                // setpoint for melt temperature control
                //--------------------------------------
                "AC".SET_MLT_1_TMP    :=    "PAR_MAIN".DI_TMP_DIPPING;

                // time till end of this step
                // --------------------------
                "APC".ACT_TME_STE := #par_time - "APC".TI[0];

                //end of step
                //-----------
                IF ("APC".TI[0] > #par_time) THEN
                    //setpoint calculation for temperature decrement
                    //----------------------------------------------
                    "AC".SET_HTR_1_TMP     :=    #htr_1_tmp_before_gap - "PAR_MAIN".DI_TMP_DEC_HTR_1;
                    #end_of_step[0] := true;
                END_IF;

                #next_step[0] := 950;


   //-step-950--level--0--------------------------------------------------------------                                                  
   //            DI: wait time after temperature decrement
   //---------------------------------------------------------------------------------                                                 
            950 :
                 IF #next_step[0] = #active_step[0] THEN   
                     "APC".TI[0] := 0;                     // start step time
                 END_IF;

                 //end of step
                 //-----------
                 IF ("APC".TI[0] > 5) THEN
                     #end_of_step[0] := true;
                 END_IF;

                 #next_step[0] := 1000;


   //-step-1000--level--0-------------------------------------------------------------                                                 
   //            DI: start neck process
   //---------------------------------------------------------------------------------                                                 
           1000 :                                                  
                 IF #next_step[0] = #active_step[0] THEN
                   "APC".OP_MSG := "OP_MSG".BLANK;
                   "DC".MOD_NE := TRUE;                           // switch to neck 
                 END_IF;

                 #next_step[0] := 1000;                        // E N D


   //-error------level--0---------------------------------------------------(error in level 0)-------------
       ELSE:                                                        
           //error code                                                //do error code
           ;        
   //------------------------------------------------------------------------------------------------------
       END_CASE;

       //check if calculated weight of grown body is changed
       //---------------------------------------------------
       IF ("KYA".CALC_WGT_GRW_XT <> #prv_calc_wgt_grw_xt) THEN
           #xt_wgt_chgd     :=  true;

       END_IF;

       //calculation length of next body
       //-------------------------------
       IF (#xt_wgt_chgd OR NOT #xt_lgh_calc_done) THEN 

           //call calculation of 2nd body length
           //-----------------------------------
           "CM_CALC_NEXT_BY" (dia            := "PAR_XT_DIA".PAR[7, 1],       
                            xt_wgt_cor     := ("KYA".CALC_WGT_GRW_XT - #prv_calc_wgt_grw_xt),
                            rm_mlt         := "CNF".RM_MLT_AFT_PRC);

           #prv_calc_wgt_grw_xt :=  "KYA".CALC_WGT_GRW_XT;
           #xt_lgh_calc_done    :=  true;
           #xt_wgt_chgd         :=  false;

       END_IF;

       #start_previous  := #start;                                   //save start input for next call 
       #cont_previous   := "APC".CONT;                                //save cont input for next call 
       #resume_previous := "APC".RESUME;                              //save resume input for next call
       #jump_previous   := "APC".JUMP;                                //save jump input for next call
       #single_previous := "APC".SINGLE;                              //save single input for next call
END_FUNCTION_BLOCK

FUNCTION_BLOCK "AM_NE"   // FB199, SCL
{ S7_Optimized_Access := 'FALSE' }
VERSION : 0.0
// --------------------------------------------------------------------------------
//     program     :    AM_NE
//     description :    apc neck module  
//     name        :    D. Bruess
//     date        :    25.11.99
// 
//     revision    :    change default rotation direction: xtal= ccw and cruc= cw
//     name        :    G. Eibelsh鋟ser
//     date        :    26.04.00
// 
//     revision    :    
//     name        :    
//     date        :    
//                     (c)CGS
//     --------------------------------------------------------------------------------
   VAR_INPUT
      start : Bool;   // start sequence, activate step 10 (impulse triggered)
   END_VAR
   VAR
      start_previous : Bool;   // start input value of last call
      cont_previous : Bool;   // cont input value of last call
      resume_previous : Bool;   // resume input value of last call
      jump_previous : Bool;   // jump input value of last call
      single_previous : Bool;   // single input value of last call
      active_step : Array[0..7] of Int;   // active step number for sequence level 0..7
      next_step : Array[0..7] of Int;   // next step number for sequence level 0..7
      hold_step : Array[0..7] of Int;   // step number of step on hold
      end_of_step : Array[0..7] of Bool;   // active step is done flag for sequence 0..7
      EndOfStep : Bool;   // default value for active step is done flag
      cont_enable : Array[0..7] of Bool;   // enable continue function
      ContEnable : Bool;   // default value for enable continue function
      ne_end : Bool;   // neck end flag
      xt_pos_at_start : Real;   // crystal position at start of neck
      xt_dia_at_start : Real;   // crystal diameter at start
      xt_dia_end_slope1 : Real;   // crystal diameter at end of slope 1
      xt_dia_end_slope2 : Real;   // crystal diameter at end of slope 2
      ini_ne_len : Real;   // initial stable neck length
   END_VAR
BEGIN


       "APC".STATUS := "APC".NECK;                                     // set apc status               

       "AM_SEQUENCE_CTL" (start_p            := #start,               // control sequence
                        start_previous_p   := #start_previous,
                        cont_previous_p    := #cont_previous, 
                        resume_previous_p  := #resume_previous,
                        jump_previous_p    := #jump_previous,
                        single_previous_p  := #single_previous,
                        active_step_p      := #active_step, 
                        next_step_p        := #next_step,
                        hold_step_p        := #hold_step, 
                        end_of_step_p      := #end_of_step, 
                        cont_enable_p      := #cont_enable); 

       //Set the "Oxidation valve" in all Phases
       "DC".V21_OP:= DINT_TO_BOOL(REAL_TO_DINT("PAR_MAIN".NE_V21_OPEN));

       CASE #active_step[0] OF    //sequence level_0
   //step--0-----level--0-------------------------------------------------off--(sequence off)--------------
           0    :                                                  
                #next_step[0] := 0;

   //step--1-----level--0-------------------------------------------------hold-(test sequence)-------------
           1   :                                                       
               IF #next_step[0] = #active_step[0] THEN                   //init step     
                   //init code
                   ; 
               END_IF;

               //step code                                             //do step
               ;

   //-step-10----level--0----------------------------------------------main-(start sequence)---------------                                                 

   //-step-10----level--0-------------------------------------------------------------                                                 
   //            NE: init neck sequence
   //---------------------------------------------------------------------------------                                                 
           10  :                                                     

               // init vacuum system
               // ------------------
               "DC".V1_OP    := TRUE;                         // open V1
               "DC".V3_OP    := FALSE;
               "DC".V4_OP    := FALSE;
               "DC".V5_OP    := TRUE;                         // open V5
               "DC".V6_OP    := FALSE;
               "DC".V8_OP    := FALSE;
               "DC".V11_OP   := FALSE;
               "DC".V11_CL   := TRUE;
               "DC".V12_OP   := FALSE;
               "DC".V13_OP   := FALSE;
               "DC".V20_OP   := FALSE;
               "DC".V22_OP   := FALSE;
               "DC".V24_OP   := FALSE;
               "DC".P1_ON    := TRUE;                         // start main pump
               "DC".P3_ON    := FALSE;
               "DC".V3_4_OP  := FALSE;
               "DC".V1_1_REL := FALSE;

               "DC".V3_2_OP := FALSE;                      // vacuum valve feeder

               "DC".V1_OPEN_REQ   := FALSE;                // only EKZ 2700
               "DC".V1_CLOSE_REQ  := FALSE;


               // init drives
               // -----------
               "DC".XT_LFT_UP := TRUE;                     // crystal lift up
               "DC".XT_LFT_DN := FALSE;
               "DC".XT_LFT_FST := FALSE;
               "DC".XT_ROT_CW := "BM_ROT_DRV_DIR_DB".ROT_DIR;            //1 = cw
               "DC".XT_ROT_CCW := NOT "BM_ROT_DRV_DIR_DB".ROT_DIR;       //0 = ccw


               "DC".CR_LFT_UP := FALSE;                    // crucible lift up
               "DC".CR_LFT_DN := FALSE;
               "DC".CR_LFT_FST := FALSE;
               "DC".CR_ROT_CW := NOT "BM_ROT_DRV_DIR_DB".ROT_DIR;        //0 = cw
               "DC".CR_ROT_CCW := "BM_ROT_DRV_DIR_DB".ROT_DIR;           //1 = ccw


               "AC".SET_XT_SPD := "KYA".SET_XT_SPD;
               "AC".SET_XT_ROT := "KYA".SET_XT_ROT;
               "AC".SET_CR_SPD := 0.0;
               "AC".SET_CR_ROT := "KYA".SET_CR_ROT;

               // init heater
               // -----------
               "DC".HTR_1_ON := TRUE;                     // heater on
               "DC".HTR_2_ON := TRUE;
               "DC".HTR_3_ON := FALSE;

               // AC.SET_HTR_1_PWR := 0.0;                 do not set, loop is on
               // AC.SET_HTR_2_PWR := 0.0;
               // AC.SET_HTR_3_PWR := 0.0;

               //mobile feeder
               //-------------
               "DC".MOB_FDR_MVE_IN_SEQ_ON    :=  FALSE;
               IF ("LT".MOB_FDR_DCK_DONE AND ("DV".FDG_MVE_IN_SEQ_DONE OR NOT "DV".FDG_MVE_OUT_SEQ_DONE)) THEN 
                   "DC".MOB_FDR_MVE_OUT_SEQ_ON   :=  TRUE;
               ELSE
                   "DC".MOB_FDR_MVE_OUT_SEQ_ON   :=  FALSE;
               END_IF;
               "DC".MOB_FDR_VIB_ON           :=  FALSE;
               "FLT".MOB_FDR_NOT_DCK         :=  FALSE;
               "FLT".MOB_FDR_STP_PARA        :=  FALSE;

               // init magnet
               // -----------
               "DC".MAG_ON := ("AC".SET_MAG_1_CUR > 0.0);                       

               "AC".SET_MAG_1_CUR := "KYA".SET_MAG_1_CUR;
               "AC".SET_MAG_2_CUR := "KYA".SET_MAG_2_CUR;

               // init control loops
               // ------------------
               "DC".CTL_DIA_ON := FALSE;                   // all control loops off
               "DC".CTL_GRW_RTE_ON := FALSE;
               "DC".CTL_PULL_RTE_ON := FALSE;
               "DC".CTL_CRUC_ROT_ON := FALSE;
               "DC".CTL_MLT_LVL_ON := FALSE;
               "DC".CTL_MLT_1_TMP_ON := FALSE;
               "DC".CTL_MLT_2_TMP_ON := FALSE;
               "DC".CTL_MLT_DRIFT_ON := FALSE;
               "DC".CTL_GAP_ON       := FALSE;
               "DC".CTL_HTR_1_TMP_ON := TRUE;              // heater temp loop on
               //  DC.CTL_HTR_2_TMP_ON := TRUE;

               "DC".SET_HTR_1_TMP_ABS := FALSE;            // enable inc functions
               "DC".SET_HTR_2_PWR_ABS := FALSE;


               "DC".CTL_PRS_ON := TRUE;                    // pressure control on

               "DC".CTL_SI_FDR_ON := FALSE;
               "DC".CTL_DOP_FDR_ON := FALSE;

               "DV".TRANS_SH_BY_FLAG := FALSE;
               "DV".START_SH_FLAG    := FALSE;

               "AC".SET_XT_DIA := 0.0;
               "AC".SET_GRW_RTE := 0.0;
               "AC".SET_AVG_SPD := 0.0;
               "AC".SET_AVG_CRUC_ROT := 0.0;
               "AC".SET_MLT_LVL_LSR := 0.0;
               "AC".SET_MLT_1_TMP := 0.0;
               "AC".SET_MLT_2_TMP := 0.0;

               // init measurement system
               // -----------------------
               "DC".CAM_ISP_ON   :=  TRUE;      //inspection on
               "DC".CAM_INIT     :=  FALSE;
               "DC".CAM_MLT      :=  FALSE;
               "DC".CAM_DIP      :=  FALSE;
               "DC".CAM_DIA      :=  TRUE;
               "DC".CAM_SEL_1    :=  TRUE;
               "DC".CAM_SEL_2    :=  FALSE;

               "DV".THR_CALC_DISABLED  := TRUE;      //threshold calculation in this step is disabled


               "DC".LSR_ON := ("PAR_MAIN".BY_LSR_LVL_CTL_ON = 1.0);    // laser on/off (parameter comes from body mode)
               "DC".MCC_ON := FALSE;                                 // melt contact control off
               "DC".MCC_TST_ON := FALSE;

               // init Si feeder system
               // ---------------------
               "DC".SI_FDR_ON := FALSE;                              // feeder off
               "DC".DOP_FDR_ON := FALSE;

               "AC".SET_FDR_SI := 0.0;
               "AC".SET_FDR_DOP := 0.0;

               // init lamp on control cabinet
               // ----------------------------
               "DV".LMP_OR := false;

               // save start position, reset length
               // ---------------------------------
               #xt_pos_at_start := "AV".ACT_XT_POS;
               "AV".ACT_XT_LEN_PRC := 0.0; 
               "AV".ACT_XT_LEN := 0.0;

               // calculate all setpoints 
               // -----------------------
               "AM_PAR_FNC_NE" (act_x_value := 0.0);
               "AC".SET_XT_DIA := "AV".ACT_XT_DIA;           // setpoint = act. diameter 

               // enable automatic mode
               // ---------------------
               "DC".MOD_AUT_ENB := TRUE;

               #end_of_step[0] := true;                            
               #next_step[0] := 100;

   //-step-100---level--0-------------------------------------------------------------                                                 
   //            NE: wait for automatic mode
   //---------------------------------------------------------------------------------                                                 
           100 :                                                     
               IF #next_step[0] = #active_step[0] THEN
                   "APC".OP_MSG := "OP_MSG".WAIT_FOR_AUTO;                                                  
               END_IF;

               // do not count the length while waiting for automatic
               // ---------------------------------------------------
               #xt_pos_at_start := "AV".ACT_XT_POS;
               "AV".ACT_XT_LEN_PRC := 0.0; 
               "AV".ACT_XT_LEN := 0.0;

               // calculate all setpoints 
               // -----------------------
               "AM_PAR_FNC_NE" (act_x_value := 0.0);
               "AC".SET_XT_DIA := "AV".ACT_XT_DIA;           // setpoint = act. diameter 

               IF "APC".AUTOMATIC = TRUE THEN                     // automatic mode ?
                   #end_of_step[0] := true;                            
               END_IF;                                    
               #next_step[0] := 200;


   //-step-200---level--0-------------------------------------------------------------                                                 
   //            NE: start time
   //---------------------------------------------------------------------------------                                                 
           200 :                                                     
               "APC".ACT_TME_PROC := 0;                           // start process time
               "APC".ACT_TME_STE := 0;                            // reset time of step
               "APC".TI[0] := 0;                                  // start waiting time
               "APC".OP_MSG := "OP_MSG".BLANK;                                                  

               //init total length calculation
               //-----------------------------
               "DV".NE_RESTART   :=  TRUE;

               #end_of_step[0] := true;                            
               #next_step[0] := 300;

   //-step-300---level--0-------------------------------------------------------------                                                 
   //            NE: do initial temp. inc. and wait (const speed, no dia. control)
   //---------------------------------------------------------------------------------                                                 
           300 :                                                     
               IF #next_step[0] = #active_step[0] THEN                       
                   //display initial temperature and power setpoints
                   //-----------------------------------------------
                   "DIS".HTR_1_TMP_SET_PHA_STR   :=  "CTL".SET_HTR_1_TMP;
                   "DIS".HTR_2_PWR_SET_PHA_STR   :=  "CTL".SET_HTR_2_PWR;
                   // do heater inc.
                   // --------------
                   "DC".RSTRT_HTR_1_TMP_INC      := TRUE;
                   "DC".RSTRT_HTR_2_PWR_INC      := TRUE;
                   "AC".SET_HTR_1_TMP_INC        := "AV".SET_HTR_1_TMP_INC;
                   "AC".SET_HTR_2_PWR_INC        := "AV".SET_HTR_2_PWR_INC;

                   "AV".SET_DIP_TMP              := "CTL".SET_HTR_1_TMP;           //store heater temp setpoint (used in removal)
                   "APC".OP_MSG                  := "OP_MSG".BY_WAIT_TILL_DIA_CTL;

               END_IF;

               // setpoint magnet
               // ---------------
               "DC".MAG_ON := ("AC".SET_MAG_1_CUR > 0.0);

               "AC".SET_MAG_1_CUR := "AV".SET_MAG_1_CUR;
               "AC".SET_MAG_2_CUR := "AV".SET_MAG_1_CUR * "AV".SET_MAG_RATIO_CUR;


               // calculate actual length
               // -----------------------
               "AM_CALC_LENGTH" (start_pos := #xt_pos_at_start,
                               actual_pos := "AV".ACT_XT_POS,
                               total_len := -1.0,              // % not calculated
                               actual_len => "AV".ACT_XT_LEN,
                               actual_len_prc => "AV".ACT_XT_LEN_PRC);


               // calculate all setpoints for this step
               // -------------------------------------                                      
               "AM_PAR_FNC_NE" (act_x_value := 0.0);
               "AC".SET_XT_DIA := "AV".ACT_XT_DIA;         // setpoint = act. diameter 
               "AC".SET_XT_SPD := "AC".SET_AVG_SPD;        // init output diam. control
               "AC".SET_HTR_1_TMP_INC := "AV".SET_HTR_1_TMP_INC;
               "AC".SET_HTR_2_PWR_INC := "AV".SET_HTR_2_PWR_INC;


               // wait time ?
               // -----------
               IF ("APC".TI[0] > 30) THEN
                  #end_of_step[0] := true;
               END_IF;

               #next_step[0] := 400; 


   //-step-400---level--0-------------------------------------------------------------                                                 
   //            NE: grow neck cone (slope 1)
   //---------------------------------------------------------------------------------                                                 
           400 :                                                  
               IF #next_step[0] = #active_step[0] THEN                       
                   // start time for slope calc.
                   // --------------------------
                   "APC".TI[0] := 0;

                   // save start diameter
                   // -------------------
                   #xt_dia_at_start := "AV".ACT_XT_DIA;
                   "AC".SET_XT_DIA   := "AV".ACT_XT_DIA;           // setpoint = act. diameter 

                   // diameter and av. speed control on
                   // ---------------------------------
                   "DC".CTL_DIA_ON       := TRUE;
                   "DC".CTL_PULL_RTE_ON  := TRUE;

                   "APC".OP_MSG := "OP_MSG".NE_DIA_REDUCTION1;
               END_IF;

               // setpoint magnet
               // ---------------
               "DC".MAG_ON := ("AC".SET_MAG_1_CUR > 0.0);

               "AC".SET_MAG_1_CUR := "AV".SET_MAG_1_CUR;
               "AC".SET_MAG_2_CUR := "AV".SET_MAG_1_CUR * "AV".SET_MAG_RATIO_CUR;

               // calculate actual length
               // -----------------------
               "AM_CALC_LENGTH" (start_pos      := #xt_pos_at_start,
                               actual_pos     := "AV".ACT_XT_POS,
                               total_len      := -1.0,              // % not calculated
                               actual_len     => "AV".ACT_XT_LEN,
                               actual_len_prc => "AV".ACT_XT_LEN_PRC);

               // calculate all setpoints for this step
               // -------------------------------------                                      
               "AM_PAR_FNC_NE" (act_x_value := 0.0);           // use first line
               #xt_dia_end_slope1 := "PAR_XT_DIA".PAR["APC".NECK, 1]
                                                  + "CNF".NECK_DELTA_SLOPE_1;
               #xt_dia_end_slope2 := "PAR_XT_DIA".PAR["APC".NECK, 1];


               "AM_CALC_NECK_DIA" (d0  := #xt_dia_at_start,
                                 dend:= #xt_dia_end_slope2,
                                 t   := INT_TO_REAL("APC".TI[0]),
                                 ddt := "CNF".NECK_SLOPE_1,
                                 dia => "AC".SET_XT_DIA);

               // heater temp/power inc.
               // ----------------------
               "AC".SET_HTR_1_TMP_INC := "AV".SET_HTR_1_TMP_INC;
               "AC".SET_HTR_2_PWR_INC := "AV".SET_HTR_2_PWR_INC;

               // melt contact control
               // --------------------   
               "DC".MCC_ON := ("PAR_MAIN".NE_MLT_CONTACT_CTL = 1.0);        


               // diameter setpoint below (final diam. + delta) ?
               // -----------------------------------------------
               IF ("AC".SET_XT_DIA < #xt_dia_end_slope1) THEN    
                   #end_of_step[0] := true;                            
               END_IF;
               #next_step[0] := 500; 


   //-step-500---level--0-------------------------------------------------------------                                                 
   //            NE: grow neck cone (slope 2)
   //---------------------------------------------------------------------------------                                                 
           500 :                                                  
               IF #next_step[0] = #active_step[0] THEN                       
                   // start time for slope calc.
                   // --------------------------
                   "APC".TI[0] := 0;

                   // save start diameter setpoint
                   // ----------------------------
                   #xt_dia_at_start := "AC".SET_XT_DIA;

                   "APC".OP_MSG := "OP_MSG".NE_DIA_REDUCTION2;
               END_IF;

               // setpoint magnet
               // ---------------
               "DC".MAG_ON := ("AC".SET_MAG_1_CUR > 0.0);

               "AC".SET_MAG_1_CUR := "AV".SET_MAG_1_CUR;
               "AC".SET_MAG_2_CUR := "AV".SET_MAG_1_CUR * "AV".SET_MAG_RATIO_CUR;


               // calculate actual length
               // -----------------------
               "AM_CALC_LENGTH" (start_pos := #xt_pos_at_start,
                               actual_pos := "AV".ACT_XT_POS,
                               total_len := -1.0,              // % not calculated
                               actual_len => "AV".ACT_XT_LEN,
                               actual_len_prc => "AV".ACT_XT_LEN_PRC);

               // calculate all setpoints for this step
               // -------------------------------------                                      
               "AM_PAR_FNC_NE" (act_x_value := 0.0);           // use first line
               #xt_dia_end_slope1 := "PAR_XT_DIA".PAR["APC".NECK, 1]
                                                  + "CNF".NECK_DELTA_SLOPE_1;
               #xt_dia_end_slope2 := "PAR_XT_DIA".PAR["APC".NECK, 1];


               "AM_CALC_NECK_DIA" (d0  := #xt_dia_at_start,
                                 dend:= #xt_dia_end_slope2,
                                 t   := INT_TO_REAL("APC".TI[0]),
                                 ddt := "CNF".NECK_SLOPE_2,
                                 dia => "AC".SET_XT_DIA);

               // heater temp/power inc.
               // ----------------------
               "AC".SET_HTR_1_TMP_INC := "AV".SET_HTR_1_TMP_INC;
               "AC".SET_HTR_2_PWR_INC := "AV".SET_HTR_2_PWR_INC;

               // melt contact control
               // --------------------   
               "DC".MCC_ON := ("PAR_MAIN".NE_MLT_CONTACT_CTL = 1.0);        

               // diameter setpoint below final diam. ?
               // -------------------------------------
               IF ("AC".SET_XT_DIA <= #xt_dia_end_slope2) THEN    
                   #end_of_step[0] := true;                            
               END_IF;
               #next_step[0] := 600; 


   //-step-600---level--0-------------------------------------------------------------                                                 
   //            NE: do neck process
   //---------------------------------------------------------------------------------                                                 
           600 :                                                  
               IF #next_step[0] = #active_step[0] THEN                       
                   // save start position, reset length
                   // ---------------------------------
                   #xt_pos_at_start := "AV".ACT_XT_POS;
                   #ini_ne_len      := 0.0;
                   "APC".OP_MSG := "OP_MSG".NE_DIA_CONSTANT;
               END_IF;

               // setpoint magnet
               // ---------------
               "DC".MAG_ON := ("AC".SET_MAG_1_CUR > 0.0);

               "AC".SET_MAG_1_CUR := "AV".SET_MAG_1_CUR;
               "AC".SET_MAG_2_CUR := "AV".SET_MAG_1_CUR * "AV".SET_MAG_RATIO_CUR;

               // heater temp/power inc.
               // ----------------------
               "AC".SET_HTR_1_TMP_INC := "AV".SET_HTR_1_TMP_INC;
               "AC".SET_HTR_2_PWR_INC := "AV".SET_HTR_2_PWR_INC;

               // melt contact control
               // --------------------   
               "DC".MCC_ON := ("PAR_MAIN".NE_MLT_CONTACT_CTL = 1.0);  

               // calculate all setpoints for this step
               // -------------------------------------                                      
               "AM_PAR_FNC_NE" (act_x_value := "AV".ACT_XT_LEN);
               "AC".SET_XT_DIA := "AV".SET_XT_DIA;


                //neck with flexible length (option)
               //----------------------------------
               IF (REAL_TO_INT("PAR_MAIN".NE_LEN_FLX) = 1) THEN  

                   // calculate actual length
                   // -----------------------
                   "AM_CALC_LENGTH" (start_pos       := #xt_pos_at_start,
                                   actual_pos      := "AV".ACT_XT_POS,
                                   total_len       := "PAR_MAIN".NE_MAX_LEN,
                                   actual_len      => "AV".ACT_XT_LEN,
                                   actual_len_prc  => "AV".ACT_XT_LEN_PRC);


                   //reset stable neck length due to diameter or growth deviation, slow pull speed or minimum neck length
                   //----------------------------------------------------------------------------------------------------
                   IF ((("AV".ACT_XT_DIA - "AC".SET_XT_DIA) > "PAR_MAIN".NE_MAX_DEV_DIA)     OR 
                       ("CTL".ACT_GRW_RTE > "PAR_MAIN".NE_MAX_DEV_LAT_GRW)                 OR
                       ("CTL".AVG_XT_SPD < "PAR_MAIN".NE_MIN_XT_SPD)                       OR 
                       ("AV".ACT_XT_LEN <= ("PAR_MAIN".NE_MIN_LEN - "PAR_MAIN".NE_STB_LEN))) THEN

                       #ini_ne_len  :=  "AV".ACT_XT_LEN;
                   END_IF;

                   //calculate stable neck length
                   //----------------------------    
                   "AV".ACT_STB_NE_LEN   :=  "AV".ACT_XT_LEN - #ini_ne_len;

                   IF ("PAR_MAIN".NE_STB_LEN > 0.0) THEN 
                       "AV".ACT_STB_NE_LEN_PRC   :=  "AV".ACT_STB_NE_LEN / "PAR_MAIN".NE_STB_LEN * 100.0;
                   END_IF;

                   //neck end when max. length is reached
                   //------------------------------------ 
                   IF  ("AV".ACT_XT_LEN >= "PAR_MAIN".NE_MAX_LEN) THEN 
                       #ne_end          :=  true;
                       "FLT".NE_MAX_LEN  :=  TRUE;

                   //neck min length reached
                   //-----------------------
                   ELSIF  ("AV".ACT_XT_LEN >= "PAR_MAIN".NE_MIN_LEN) THEN 
                       //check stable neck length
                       //------------------------
                       IF ("AV".ACT_STB_NE_LEN >= "PAR_MAIN".NE_STB_LEN) THEN
                           #ne_end  :=  true;
                       ELSE
                           #ne_end  :=  false;
                       END_IF;
                   ELSE
                       #ne_end  :=  false;
                   END_IF;

                   // check if neck end is reached ?
                   // ------------------------------
                   IF #ne_end THEN    
                       #end_of_step[0] := true;                            
                   END_IF;

               //neck with fixed length (standard)
               //---------------------------------
               ELSE 

                   // calculate actual length
                   // -----------------------
                   "AM_CALC_LENGTH" (start_pos       := #xt_pos_at_start,
                                   actual_pos      := "AV".ACT_XT_POS,
                                   total_len       := "PAR_MAIN".NE_LEN,
                                   actual_len      => "AV".ACT_XT_LEN,
                                   actual_len_prc  => "AV".ACT_XT_LEN_PRC);

                   // 100% of length reached ?
                   // ------------------------
                   IF ("AV".ACT_XT_LEN_PRC >= 100.0) THEN    
                       #end_of_step[0] := true;                            
                   END_IF;

               END_IF;
               #next_step[0] := 700; 


   //-step-700---level--0-------------------------------------------------------------                                                 
   //            NE: start shoulder process
   //---------------------------------------------------------------------------------                                                 
           700 :                                                  
               IF #next_step[0] = #active_step[0] THEN
                   "APC".OP_MSG := "OP_MSG".BLANK;
               END_IF;

               "DC".MOD_SH := TRUE;                               // switch to shoulder 
               #next_step[0] := 700;                             // E N D 



   //-error------level--0---------------------------------------------------(error in level 0)-------------
       ELSE:                                                        
           //error code                                                //do error code
           ;        
   //------------------------------------------------------------------------------------------------------
       END_CASE;

       CASE #active_step[1] OF    //sequence level_1
   //step--0-----level--1-------------------------------------------------off--(sequence off)--------------
           0    :                                                  
                #next_step[1] := 0;

   //step--1-----level--1-------------------------------------------------hold-(test sequence)-------------
           1   :                                                       
               IF #next_step[1] = #active_step[1] THEN                   //init step     
                   //init code
                   ; 
               END_IF;

               //step code                                             //do step
               ;

   //-step-10----level--1----------------------------------------------main-(start sequence)---------------                                                 
           10  :                                                     
               IF #next_step[1] = #active_step[1] THEN                   //init step     
                   //init code 
                   ;                                                  
               END_IF;

               //step code                                             //do step
               ;
               IF #ContEnable = true THEN                               //enable continue function
                   #cont_enable[1] := true;
               END_IF;
               IF #EndOfStep = true THEN                                //define end of step condition
                   #end_of_step[1] := true;                            
               END_IF;                                    
               #next_step[1] := 0;                                      //define next step #
               IF #end_of_step[1] = true THEN                           //do on transition
                   //transition code
                   ;
               END_IF;

   //-step-100---level--1----------------------------------------------name-(remarks)----------------------                                                 
           100 :                                                     
               IF #next_step[1] = #active_step[1] THEN                   //init step     
                   //init code 
                   ;                                                  
               END_IF;

               //step code                                             //do step
               ;
               IF #ContEnable = true THEN                               //enable continue function
                   #cont_enable[1] := true;
               END_IF;
               IF #EndOfStep = true THEN                                //define end of step condition
                   #end_of_step[1] := true;                            
               END_IF;                                    
               #next_step[1] := 0;                                      //define next step #
               IF #end_of_step[1] = true THEN                           //do on transition
                   //transition code
                   ;
               END_IF;

   //-step-200---level--1----------------------------------------------name-(remarks)----------------------                                                 
           200 :                                                     
               IF #next_step[1] = #active_step[1] THEN                   //init step     
                   //init code 
                   ;                                                  
               END_IF;

               //step code                                             //do step
               ;
               IF #ContEnable = true THEN                               //enable continue function
                   #cont_enable[1] := true;
               END_IF;
               IF #EndOfStep = true THEN                                //define end of step condition
                   #end_of_step[1] := true;                            
               END_IF;                                    
               #next_step[1] := 0;                                      //define next step #
               IF #end_of_step[1] = true THEN                           //do on transition
                   //transition code
                   ;
               END_IF;

   //-error------level--1---------------------------------------------------(error in level 1)-------------
       ELSE:                                                        
           //error code                                                //do error code
           ;        
   //------------------------------------------------------------------------------------------------------
       END_CASE;

       CASE #active_step[2] OF    //sequence level_2
   //step--0-----level--2-------------------------------------------------off--(sequence off)--------------
           0    :                                                  
                #next_step[2] := 0;

   //step--1-----level--2-------------------------------------------------hold-(test sequence)-------------
           1   :                                                       
               IF #next_step[2] = #active_step[2] THEN                   //init step     
                   //init code
                   ; 
               END_IF;

               //step code                                             //do step
               ;

   //-step-10----level--2----------------------------------------------main-(start sequence)---------------                                                 
           10  :                                                     
               IF #next_step[2] = #active_step[2] THEN                   //init step     
                   //init code 
                   ;                                                  
               END_IF;

               //step code                                             //do step
               ;
               IF #ContEnable = true THEN                               //enable continue function
                   #cont_enable[2] := true;
               END_IF;
               IF #EndOfStep = true THEN                                //define end of step condition
                   #end_of_step[2] := true;                            
               END_IF;                                    
               #next_step[1] := 0;                                      //define next step #
               IF #end_of_step[2] = true THEN                           //do on transition
                   //transition code
                   ;
               END_IF;

   //-step-100---level--2----------------------------------------------name-(remarks)----------------------                                                 
           100 :                                                     
               IF #next_step[2] = #active_step[2] THEN                   //init step     
                   //init code 
                   ;                                                  
               END_IF;

               //step code                                             //do step
               ;
               IF #ContEnable = true THEN                               //enable continue function
                   #cont_enable[2] := true;
               END_IF;
               IF #EndOfStep = true THEN                                //define end of step condition
                   #end_of_step[2] := true;                            
               END_IF;                                    
               #next_step[2] := 0;                                      //define next step #
               IF #end_of_step[2] = true THEN                           //do on transition
                   //transition code
                   ;
               END_IF;

   //-error------level--2---------------------------------------------------(error in level 2)-------------
       ELSE:                                                        
           //error code                                                //do error code
           ;        
   //------------------------------------------------------------------------------------------------------
       END_CASE;

       #start_previous := #start;                                    //save start input for next call 
       #cont_previous := "APC".CONT;                                  //save cont input for next call 
       #resume_previous := "APC".RESUME;                              //save resume input for next call
       #jump_previous := "APC".JUMP;                                  //save jump input for next call
       #single_previous := "APC".SINGLE;                              //save single input for next call
END_FUNCTION_BLOCK

FUNCTION_BLOCK "AM_SH"   // FB200, SCL
{ S7_Optimized_Access := 'FALSE' }
VERSION : 0.0
// --------------------------------------------------------------------------------
//     program     :    AM_SH
//     description :    apc shoulder module  
//     name        :    D. Bruess
//     date        :    30.11.99
// 
//     revision    :    change default rotation direction: xtal= ccw and cruc= cw
//     name        :    G. Eibelsh鋟ser
//     date        :    26.04.00
// 
//     revision    :    
//     name        :    
//     date        :    
//                     (c)CGS
//     --------------------------------------------------------------------------------
   VAR_INPUT
      start : Bool;   // start sequence, activate step 10 (impulse triggered)
   END_VAR
   VAR
      start_previous : Bool;   // start input value of last call
      cont_previous : Bool;   // cont input value of last call
      resume_previous : Bool;   // resume input value of last call
      jump_previous : Bool;   // jump input value of last call
      single_previous : Bool;   // single input value of last call
      active_step : Array[0..7] of Int;   // active step number for sequence level 0..7
      next_step : Array[0..7] of Int;   // next step number for sequence level 0..7
      hold_step : Array[0..7] of Int;   // step number of step on hold
      end_of_step : Array[0..7] of Bool;   // active step is done flag for sequence 0..7
      EndOfStep : Bool;   // default value for active step is done flag
      cont_enable : Array[0..7] of Bool;   // enable continue function
      ContEnable : Bool;   // default value for enable continue function
      xt_pos_at_start : Real;   // crystal position at start of neck
      xt_dia_at_start : Real;   // crystal diameter at start
      xt_dia_end_slope1 : Real;   // crystal diameter at end of slope 1
      xt_dia_end_slope2 : Real;   // crystal diameter at end of slope 2
      temp1_before_gap : Real;   // heater temp1 before temp gap
   END_VAR
BEGIN


       "APC".STATUS := "APC".SHOULDER;                                 // set apc status               

       "AM_SEQUENCE_CTL" (start_p            := #start,               // control sequence
                        start_previous_p   := #start_previous,
                        cont_previous_p    := #cont_previous, 
                        resume_previous_p  := #resume_previous,
                        jump_previous_p    := #jump_previous,
                        single_previous_p  := #single_previous,
                        active_step_p      := #active_step, 
                        next_step_p        := #next_step,
                        hold_step_p        := #hold_step, 
                        end_of_step_p      := #end_of_step, 
                        cont_enable_p      := #cont_enable); 

       //Set the "Oxidation valve" in all Phases
       "DC".V21_OP:= DINT_TO_BOOL(REAL_TO_DINT("PAR_MAIN".SH_V21_OPEN));

       CASE #active_step[0] OF    //sequence level_0
   //step--0-----level--0-------------------------------------------------off--(sequence off)--------------
           0    :                                                  
                #next_step[0] := 0;

   //step--1-----level--0-------------------------------------------------hold-(test sequence)-------------
           1   :                                                       
               IF #next_step[0] = #active_step[0] THEN                   //init step     
                   //init code
                   ; 
               END_IF;

               //step code                                             //do step
               ;

   //-step-10----level--0----------------------------------------------main-(start sequence)---------------                                                 

   //-step-10----level--0-------------------------------------------------------------                                                 
   //            SH: init shoulder sequence
   //---------------------------------------------------------------------------------                                                 
           10  :                                                     

               // init vacuum system
               // ------------------
               "DC".V1_OP    := TRUE;                         // open V1
               "DC".V3_OP    := FALSE;
               "DC".V4_OP    := FALSE;
               "DC".V5_OP    := TRUE;                         // open V5
               "DC".V6_OP    := FALSE;
               "DC".V8_OP    := FALSE;
               "DC".V11_OP   := FALSE;
               "DC".V11_CL   := TRUE;
               "DC".V12_OP   := FALSE;
               "DC".V13_OP   := FALSE;
               "DC".V20_OP   := FALSE;
               "DC".V22_OP   := FALSE;
               "DC".V24_OP   := FALSE;
               "DC".P1_ON    := TRUE;                         // start main pump
               "DC".P3_ON    := FALSE;
               "DC".V3_4_OP  := FALSE;
               "DC".V1_1_REL := FALSE;

               "DC".V1_OPEN_REQ   := FALSE;                // only EKZ 2700
               "DC".V1_CLOSE_REQ  := FALSE;

               "DC".V3_2_OP := FALSE;                      // vacuum valve feeder

               // init drives
               // -----------
               "DC".XT_LFT_UP := TRUE;                     // crystal lift up
               "DC".XT_LFT_DN := FALSE;
               "DC".XT_LFT_FST := FALSE;
               "DC".XT_ROT_CW := "BM_ROT_DRV_DIR_DB".ROT_DIR;            //1 = cw
               "DC".XT_ROT_CCW := NOT "BM_ROT_DRV_DIR_DB".ROT_DIR;       //0 = ccw


               "DC".CR_LFT_UP := TRUE;                     // crucible lift up
               "DC".CR_LFT_DN := FALSE;
               "DC".CR_LFT_FST := FALSE;
               "DC".CR_ROT_CW := NOT "BM_ROT_DRV_DIR_DB".ROT_DIR;        //0 = cw
               "DC".CR_ROT_CCW := "BM_ROT_DRV_DIR_DB".ROT_DIR;           //1 = ccw


               "AC".SET_XT_SPD := "KYA".SET_XT_SPD;                
               "AC".SET_XT_ROT := "KYA".SET_XT_ROT;
               "AC".SET_CR_SPD := "KYA".SET_CR_SPD;
               "AC".SET_CR_ROT := "KYA".SET_CR_ROT;


               // init heater
               // -----------
               "DC".HTR_1_ON := TRUE;                     // heater on
               "DC".HTR_2_ON := TRUE;
               "DC".HTR_3_ON := FALSE;

               // AC.SET_HTR_1_PWR := 0.0;                 do not set, loop is on
               // AC.SET_HTR_2_PWR := 0.0;
               // AC.SET_HTR_3_PWR := 0.0;

               //mobile feeder
               //-------------
               "DC".MOB_FDR_MVE_IN_SEQ_ON    :=  FALSE;
               IF ("LT".MOB_FDR_DCK_DONE AND ("DV".FDG_MVE_IN_SEQ_DONE OR NOT "DV".FDG_MVE_OUT_SEQ_DONE)) THEN 
                   "DC".MOB_FDR_MVE_OUT_SEQ_ON   :=  TRUE;
               ELSE
                   "DC".MOB_FDR_MVE_OUT_SEQ_ON   :=  FALSE;
               END_IF;
               "DC".MOB_FDR_VIB_ON           :=  FALSE;
               "FLT".MOB_FDR_NOT_DCK         :=  FALSE;
               "FLT".MOB_FDR_STP_PARA        :=  FALSE;

               // init magnet
               // -----------
               "DC".MAG_ON := ("AC".SET_MAG_1_CUR > 0.0);                    // magnet on

               "AC".SET_MAG_1_CUR := "KYA".SET_MAG_1_CUR;
               "AC".SET_MAG_2_CUR := "KYA".SET_MAG_1_CUR * "KYA".SET_MAG_RATIO_CUR;

               // init control loops
               // ------------------
               "DC".CTL_DIA_ON       := FALSE;             // all control loops off
               "DC".CTL_GRW_RTE_ON   := FALSE;
               "DC".CTL_PULL_RTE_ON  := FALSE;
               "DC".CTL_CRUC_ROT_ON := FALSE;
               "DC".CTL_MLT_LVL_ON   := TRUE;              // for ratio calc.
               "DC".CTL_MLT_1_TMP_ON := FALSE;
               "DC".CTL_MLT_2_TMP_ON := FALSE;
               "DC".CTL_MLT_DRIFT_ON := FALSE;
               "DC".CTL_GAP_ON       := FALSE;

               "DC".CTL_HTR_1_TMP_ON := TRUE;              // heater temp loop on
               //  DC.CTL_HTR_2_TMP_ON := TRUE;

               "DC".SET_HTR_1_TMP_ABS := FALSE;            // enable inc functions
               "DC".SET_HTR_2_PWR_ABS := FALSE;


               "DC".CTL_PRS_ON := TRUE;                    // pressure control on

               "DC".CTL_SI_FDR_ON := FALSE;
               "DC".CTL_DOP_FDR_ON := FALSE;

               "AC".SET_XT_DIA := 0.0;
               "AC".SET_GRW_RTE := 0.0;
               "AC".SET_AVG_SPD := 0.0;
               "AC".SET_AVG_CRUC_ROT := 0.0;
               "AC".SET_MLT_1_TMP := 0.0;
               "AC".SET_MLT_2_TMP := 0.0;

               IF ("PAR_MAIN".BY_LSR_LVL_CTL_ON = 1.0) AND "CNF".CONF_LSR_LVL  THEN
                   "AV".SET_MLT_LVL_LSR  := "CTL".ACT_MLT_LVL; //setpoint melt level is written with actual signal of melt level
               ELSE
                   "AV".SET_MLT_LVL_LSR  := 0.0;
               END_IF;    
               "AC".SET_MLT_LVL_LSR  := "AV".SET_MLT_LVL_LSR;

               // init measurement system
               // -----------------------
               "DC".CAM_ISP_ON   :=  TRUE;      //inspection on
               "DC".CAM_INIT     :=  FALSE;
               "DC".CAM_MLT      :=  FALSE;
               "DC".CAM_DIP      :=  FALSE;
               "DC".CAM_DIA      :=  TRUE;
               "DC".CAM_SEL_1    :=  TRUE;
               "DC".CAM_SEL_2    :=  FALSE;

               "DV".THR_CALC_DISABLED  := TRUE;      //threshold calculation in this step is disabled

               "DC".LSR_ON := ("PAR_MAIN".BY_LSR_LVL_CTL_ON = 1.0);    // laser on/off (parameter comes from body mode)                             
               "DC".MCC_TST_ON := FALSE;
               "DC".MCC_ON := FALSE;                       // melt contact control off
               // init Si feeder system
               // ---------------------
               "DC".SI_FDR_ON := FALSE;                              // feeder off
               "DC".DOP_FDR_ON := FALSE;

               "AC".SET_FDR_SI := 0.0;
               "AC".SET_FDR_DOP := 0.0;

               // init lamp on control cabinet
               // ----------------------------
               "DV".LMP_OR := false;

               // save start position, reset length
               // ---------------------------------
               #xt_pos_at_start := "AV".ACT_XT_POS;
               "AV".ACT_XT_LEN_PRC := 0.0; 
               "AV".ACT_XT_LEN := 0.0;

               // init status flags
               //------------------
               "DV".START_SH_FLAG    := TRUE;
               "DV".TRANS_SH_BY_FLAG := FALSE;

               //init Si charge weight calculation
               //----------------------------------
               "DV".NEW_SI_CRG_WGT_CALC :=  TRUE;

               // calculate all setpoints 
               // -----------------------
               IF "CNF".CONF_SH_PAR_FNCT = TRUE  THEN
                   "AM_PAR_FNC_SH" (act_x_value := "AV".ACT_XT_LEN);        //use shoulder parameters as function of length
               ELSE    
                   "AM_PAR_FNC_SH" (act_x_value := "AV".ACT_XT_DIA);        //use shoulder parameters as function of diameter
               END_IF;    

               // enable automatic mode
               // ---------------------
               "DC".MOD_AUT_ENB := TRUE;

               #end_of_step[0] := true;                            
               #next_step[0] := 100;


   //-step-100---level--0-------------------------------------------------------------                                                 
   //            SH: wait for automatic mode
   //---------------------------------------------------------------------------------                                                 
           100 :                                                     
               IF #next_step[0] = #active_step[0] THEN
                   "APC".OP_MSG := "OP_MSG".WAIT_FOR_AUTO;                                                  
               END_IF;

               // do not count the length while waiting for automatic
               // ---------------------------------------------------
               #xt_pos_at_start := "AV".ACT_XT_POS;
               "AV".ACT_XT_LEN_PRC := 0.0; 
               "AV".ACT_XT_LEN := 0.0;

               // calculate ratio
               // ---------------
               "AV".CRUC_RATIO := "CM_CRUC_RATIO_SH"();

               // calculate all setpoints 
               // -----------------------
               IF "CNF".CONF_SH_PAR_FNCT = TRUE  THEN
                   "AM_PAR_FNC_SH" (act_x_value := "AV".ACT_XT_LEN);        //use shoulder parameters as function of length
               ELSE    
                   "AM_PAR_FNC_SH" (act_x_value := "AV".ACT_XT_DIA);        //use shoulder parameters as function of diameter
               END_IF;    

               IF "APC".AUTOMATIC = TRUE THEN                     // automatic mode ?
                   #end_of_step[0] := true;                            
               END_IF;                                    
               #next_step[0] := 200;


   //-step-200---level--0-------------------------------------------------------------                                                 
   //            SH: start time
   //---------------------------------------------------------------------------------                                                 
           200 :                                                     
               "APC".ACT_TME_PROC := 0;                           // start process time
               "APC".ACT_TME_STE := 0;                            // reset time of step
               "APC".TI[0] := 0;                                  // start waiting time
               "APC".OP_MSG := "OP_MSG".BLANK;                                                  

               #end_of_step[0] := true;                            
               #next_step[0] := 300;


   //-step-300---level--0-------------------------------------------------------------                                                 
   //            SH: do initial temp. inc.
   //---------------------------------------------------------------------------------                                                 
           300 :                                                     
               IF #next_step[0] = #active_step[0] THEN                       
                   //display initial temperature and power setpoints
                   //-----------------------------------------------
                   "DIS".HTR_1_TMP_SET_PHA_STR   :=  "CTL".SET_HTR_1_TMP;
                   "DIS".HTR_2_PWR_SET_PHA_STR   :=  "CTL".SET_HTR_2_PWR;
                   // do heater inc.
                   // --------------
                   "DC".RSTRT_HTR_1_TMP_INC := TRUE;
                   "DC".RSTRT_HTR_2_PWR_INC := TRUE;
                   "AC".SET_HTR_1_TMP_INC := "AV".SET_HTR_1_TMP_INC;
                   "AC".SET_HTR_2_PWR_INC := "AV".SET_HTR_2_PWR_INC;
               END_IF;

               // calculate actual length
               // -----------------------
               "AM_CALC_LENGTH" (start_pos := #xt_pos_at_start,
                               actual_pos := "AV".ACT_XT_POS,
                               total_len := -1.0,
                               actual_len => "AV".ACT_XT_LEN,
                               actual_len_prc => "AV".ACT_XT_LEN_PRC);

               // calculate ratio
               // ---------------
               "AV".CRUC_RATIO := "CM_CRUC_RATIO_SH"();


               // calculate all setpoints 
               // -----------------------
               IF "CNF".CONF_SH_PAR_FNCT = TRUE  THEN
                   "AM_PAR_FNC_SH" (act_x_value := "AV".ACT_XT_LEN);        //use shoulder parameters as function of length
               ELSE    
                   "AM_PAR_FNC_SH" (act_x_value := "AV".ACT_XT_DIA);        //use shoulder parameters as function of diameter
               END_IF;    

               // setpoint magnet
               // ---------------
               "DC".MAG_ON := ("AC".SET_MAG_1_CUR > 0.0);

               "AC".SET_MAG_1_CUR := "AV".SET_MAG_1_CUR;
               "AC".SET_MAG_2_CUR := "AV".SET_MAG_1_CUR * "AV".SET_MAG_RATIO_CUR;

               //calculate setpoint melt level
               //-----------------------------
               IF ("PAR_MAIN".BY_LSR_LVL_CTL_ON = 1.0) AND "CNF".CONF_LSR_LVL  THEN
                   "AC".SET_MLT_LVL_LSR  := "AV".SET_MLT_LVL_LSR + "AC".SET_MLT_LVL_INC;
               END_IF;    

               #end_of_step[0] := true;
               #next_step[0] := 400; 


   //-step-400---level--0-------------------------------------------------------------                                                 
   //            SH: temperature gap for one 60 sec
   //---------------------------------------------------------------------------------                                                 
           400 :                                                  
               IF #next_step[0] = #active_step[0] THEN

                   // dec. temp for temp. gap
                   // -----------------------
                   #temp1_before_gap :="AV".SET_HTR_1_TMP_INC;
                   "AC".SET_HTR_1_TMP_INC := #temp1_before_gap - 
                                               "PAR_MAIN".SH_TMP_GAP_HTR_1;

                   // start time for temperature gap
                   // ------------------------------
                   "APC".OP_MSG := "OP_MSG".BLANK;
                   "APC".TI[0] := 0;
               END_IF;

               // time till end of temp. gap
               // --------------------------
               "APC".ACT_TME_STE := 60 - "APC".TI[0];

               // calculate actual length
               // -----------------------
               "AM_CALC_LENGTH" (start_pos      := #xt_pos_at_start,
                               actual_pos     := "AV".ACT_XT_POS,
                               total_len      := -1.0,
                               actual_len     => "AV".ACT_XT_LEN,
                               actual_len_prc => "AV".ACT_XT_LEN_PRC);

               // calculate ratio
               // ---------------
               "AV".CRUC_RATIO := "CM_CRUC_RATIO_SH"();

               // calculate all setpoints 
               // -----------------------
               IF "CNF".CONF_SH_PAR_FNCT = TRUE  THEN
                   "AM_PAR_FNC_SH" (act_x_value := "AV".ACT_XT_LEN);        //use shoulder parameters as function of length
               ELSE    
                   "AM_PAR_FNC_SH" (act_x_value := "AV".ACT_XT_DIA);        //use shoulder parameters as function of diameter
               END_IF;    

               // setpoint magnet
               // ---------------
               "DC".MAG_ON := ("AC".SET_MAG_1_CUR > 0.0);

               "AC".SET_MAG_1_CUR := "AV".SET_MAG_1_CUR;
               "AC".SET_MAG_2_CUR := "AV".SET_MAG_2_CUR * "AV".SET_MAG_RATIO_CUR;

               //calculate setpoint melt level
               //-----------------------------
               IF ("PAR_MAIN".BY_LSR_LVL_CTL_ON = 1.0) AND "CNF".CONF_LSR_LVL  THEN
                   "AC".SET_MLT_LVL_LSR  := "AV".SET_MLT_LVL_LSR + "AC".SET_MLT_LVL_INC;
               END_IF;    

               // gap time reached ?
               // ------------------
               IF ("APC".TI[0] > 60) THEN

                   // restore old temperature
                   // -----------------------
                   "AC".SET_HTR_1_TMP_INC := #temp1_before_gap;

                   #end_of_step[0] := true;                            
               END_IF;
               #next_step[0] := 500; 


   //-step-500---level--0-------------------------------------------------------------                                                 
   //            SH: wait till growth control on (180 sec)
   //---------------------------------------------------------------------------------                                                 
           500 :                                                  
               IF #next_step[0] = #active_step[0] THEN                       
                   // start wait time
                   // ---------------
                   "APC".OP_MSG := "OP_MSG".SH_WAIT_TILL_GROWTH_CTL;
                   "APC".TI[0] := 0;
               END_IF;

               // time till end of wait time
               // --------------------------
               "APC".ACT_TME_STE := 180 - "APC".TI[0];

               // calculate actual length
               // -----------------------
               "AM_CALC_LENGTH" (start_pos := #xt_pos_at_start,
                               actual_pos := "AV".ACT_XT_POS,
                               total_len := -1.0,
                               actual_len => "AV".ACT_XT_LEN,
                               actual_len_prc => "AV".ACT_XT_LEN_PRC);

               // calculate ratio
               // ---------------
               "AV".CRUC_RATIO := "CM_CRUC_RATIO_SH"();

               // calculate all setpoints 
               // -----------------------
               IF "CNF".CONF_SH_PAR_FNCT = TRUE  THEN
                   "AM_PAR_FNC_SH" (act_x_value := "AV".ACT_XT_LEN);        //use shoulder parameters as function of length
               ELSE    
                   "AM_PAR_FNC_SH" (act_x_value := "AV".ACT_XT_DIA);        //use shoulder parameters as function of diameter
               END_IF;    

               // setpoint magnet
               // ---------------
               "DC".MAG_ON := ("AC".SET_MAG_1_CUR > 0.0);

               "AC".SET_MAG_1_CUR := "AV".SET_MAG_1_CUR;
               "AC".SET_MAG_2_CUR := "AV".SET_MAG_1_CUR * "AV".SET_MAG_RATIO_CUR;

               //calculate setpoint melt level
               //-----------------------------
               IF ("PAR_MAIN".BY_LSR_LVL_CTL_ON = 1.0) AND "CNF".CONF_LSR_LVL  THEN
                   "AC".SET_MLT_LVL_LSR  := "AV".SET_MLT_LVL_LSR + "AC".SET_MLT_LVL_INC;
               END_IF;    

               // heater temp/power inc.
               // ----------------------
               "AC".SET_HTR_1_TMP_INC := "AV".SET_HTR_1_TMP_INC;
               "AC".SET_HTR_2_PWR_INC := "AV".SET_HTR_2_PWR_INC;

               // wait time reached ?
               // -------------------
               IF ("APC".TI[0] > 180) THEN    
                   #end_of_step[0] := true;                            
               END_IF;
               #next_step[0] := 600; 


   //-step-600---level--0-------------------------------------------------------------                                                 
   //            SH: shoulder with growth control
   //---------------------------------------------------------------------------------                                                 
           600 :                                                  
               IF #next_step[0] = #active_step[0] THEN                       
                   // switch growth control on
                   // ------------------------
                   "APC".OP_MSG := "OP_MSG".SH_WITH_GROWTH_CTL;
                   "APC".ACT_TME_STE     := 0;
                   "DC".CTL_GRW_RTE_ON   := TRUE;
                   "DV".START_SH_FLAG    := FALSE;
                   "FLT".NE_MAX_LEN      := FALSE;   //reset "max neck length reached" alarm
               END_IF;

               //set crucible rotation controller
               //--------------------------------
               "DC".CTL_CRUC_ROT_ON  := "PAR_MAIN".SH_CRUC_ROT_CTL_ON = 1.0;

               // calculate actual length
               // -----------------------
               "AM_CALC_LENGTH" (start_pos := #xt_pos_at_start,
                               actual_pos := "AV".ACT_XT_POS,
                               total_len := -1.0,
                               actual_len => "AV".ACT_XT_LEN,
                               actual_len_prc => "AV".ACT_XT_LEN_PRC);

               // calculate ratio
               // ---------------
               "AV".CRUC_RATIO := "CM_CRUC_RATIO_SH"();

               // calculate all setpoints 
               // -----------------------
               IF "CNF".CONF_SH_PAR_FNCT = TRUE  THEN
                   "AM_PAR_FNC_SH" (act_x_value := "AV".ACT_XT_LEN);        //use shoulder parameters as function of length
               ELSE    
                   "AM_PAR_FNC_SH" (act_x_value := "AV".ACT_XT_DIA);        //use shoulder parameters as function of diameter
               END_IF;    

               // setpoint magnet
               // ---------------
               "DC".MAG_ON := ("AC".SET_MAG_1_CUR > 0.0);

               "AC".SET_MAG_1_CUR := "AV".SET_MAG_1_CUR;
               "AC".SET_MAG_2_CUR := "AV".SET_MAG_2_CUR * "AV".SET_MAG_RATIO_CUR;

               //calculate setpoint melt level
               //-----------------------------
               IF ("PAR_MAIN".BY_LSR_LVL_CTL_ON = 1.0) AND "CNF".CONF_LSR_LVL  THEN
                   "AC".SET_MLT_LVL_LSR  := "AV".SET_MLT_LVL_LSR + "AC".SET_MLT_LVL_INC;
               END_IF;    

               // heater temp/power inc.
               // ----------------------
               "AC".SET_HTR_1_TMP_INC := "AV".SET_HTR_1_TMP_INC;
               "AC".SET_HTR_2_PWR_INC := "AV".SET_HTR_2_PWR_INC;

               //start transition to body with flexible diameter (option)
               //--------------------------------------------------------
               IF (REAL_TO_INT("PAR_MAIN".SH_TRS_FLX) = 1) THEN 
                   //calculate shoulder diameter for start of transition
                   //---------------------------------------------------
                   IF ("CTL".ACT_GRW_RTE >= 0.0) THEN 
                       "AV".SH_TRS_DIA   :=  "PAR_MAIN".SH_COEFFICIENT_A + "PAR_MAIN".SH_COEFFICIENT_B * "CTL".ACT_GRW_RTE;
                   END_IF;

                   //transition start when max. diameter is reached
                   //----------------------------------------------
                   IF  ("AV".ACT_XT_DIA >= "PAR_MAIN".SH_BY_TRS_MAX_DIA) THEN 
                       #end_of_step[0] := true;  

                   //transition start when when calculated transition diameter is reached
                   //--------------------------------------------------------------------
                   ELSIF ("AV".ACT_XT_DIA >= "AV".SH_TRS_DIA) THEN    
                       #end_of_step[0] := true;                            

                   END_IF;

               //start transition to body at fixed diameter (standard)
               //-----------------------------------------------------
               ELSE
                   // transition diameter reached ?
                   // -----------------------------
                   IF ("AV".ACT_XT_DIA >= "PAR_MAIN".SH_BODY_TRANS_DIA) THEN    
                       #end_of_step[0] := true;                            
                   END_IF;
               END_IF;

               #next_step[0] := 700; 

   //-step-700---level--0-------------------------------------------------------------                                                 
   //            SH: transition cycle (without growth control)
   //---------------------------------------------------------------------------------                                                 
           700 :                                                  
               IF #next_step[0] = #active_step[0] THEN                       
                   // switch growth control off
                   // -------------------------
                   "APC".OP_MSG := "OP_MSG".SH_TRANSITION_TO_BODY;
                   "DC".CTL_GRW_RTE_ON   := FALSE;
                   "DC".CTL_CRUC_ROT_ON  := FALSE;
                   "DV".TRANS_SH_BY_FLAG := TRUE;
                   "APC".TI[0] := 0;
                   "APC".TI[1] := 0;
               END_IF;

               // calculate actual length
               // -----------------------
               "AM_CALC_LENGTH" (start_pos := #xt_pos_at_start,
                               actual_pos := "AV".ACT_XT_POS,
                               total_len := -1.0,
                               actual_len => "AV".ACT_XT_LEN,
                               actual_len_prc => "AV".ACT_XT_LEN_PRC);

               // calculate ratio
               // ---------------
               "AV".CRUC_RATIO := "CM_CRUC_RATIO_SH"();

               // calculate all setpoints 
               // -----------------------
               IF "CNF".CONF_SH_PAR_FNCT = TRUE  THEN
                   "AM_PAR_FNC_SH" (act_x_value := "AV".ACT_XT_LEN);        //use shoulder parameters as function of length
               ELSE    
                   "AM_PAR_FNC_SH" (act_x_value := "AV".ACT_XT_DIA);        //use shoulder parameters as function of diameter
               END_IF;    

               // setpoint magnet
               // ---------------
               "DC".MAG_ON := ("AC".SET_MAG_1_CUR > 0.0);

               "AC".SET_MAG_1_CUR := "AV".SET_MAG_1_CUR;
               "AC".SET_MAG_2_CUR := "AV".SET_MAG_1_CUR * "AV".SET_MAG_RATIO_CUR;;

               //calculate setpoint melt level
               //-----------------------------
               IF ("PAR_MAIN".BY_LSR_LVL_CTL_ON = 1.0) AND "CNF".CONF_LSR_LVL  THEN
                   "AC".SET_MLT_LVL_LSR  := "AV".SET_MLT_LVL_LSR + "AC".SET_MLT_LVL_INC;
               END_IF;    

               // heater temp/power inc.
               // ----------------------
               "AC".SET_HTR_1_TMP_INC := "AV".SET_HTR_1_TMP_INC;
               "AC".SET_HTR_2_PWR_INC := "AV".SET_HTR_2_PWR_INC;

               (*
               // diameter for start body reached ?
               // ---------------------------------
               IF (AV.ACT_XT_DIA >= PAR_MAIN.SH_BODY_START_DIA) THEN    
                   end_of_step[0] := true;                            
               END_IF;
               *)

               //transistion to body growth reached?
               //-----------------------------------
               IF ("APC".TI[1] >= 120) THEN 
                   IF ("CTL".ACT_GRW_RTE <= "PAR_MAIN".SH_BODY_TRANS_GRW)  THEN
                       IF ("APC".TI[0] >= (REAL_TO_INT("PAR_MAIN".SH_BODY_TRANS_DLY_TME))) THEN  //delay switching to body
                           #end_of_step[0] := true;
                       END_IF;
                   ELSE
                       "APC".TI[0] := 0;
                   END_IF;
               ELSE 
                   "APC".TI[0] := 0;
               END_IF;

               #next_step[0] := 800; 

   //-step-800---level--0-------------------------------------------------------------                                                 
   //            SH: start body process
   //---------------------------------------------------------------------------------                                                 
           800 :                                                  
               IF #next_step[0] = #active_step[0] THEN
                   "APC".OP_MSG := "OP_MSG".BLANK;
               END_IF;

               "DC".MOD_BY := TRUE;                               // switch to body 
               #next_step[0] := 800;                             // E N D 



   //---------------------------------------------------------------------------------                                                 
   //-error------level--0---------------------------------------------------(error in level 0)-------------
       ELSE:                                                        
           //error code                                                //do error code
           ;        
   //------------------------------------------------------------------------------------------------------
       END_CASE;


       #start_previous := #start;                                    //save start input for next call 
       #cont_previous := "APC".CONT;                                  //save cont input for next call 
       #resume_previous := "APC".RESUME;                              //save resume input for next call
       #jump_previous := "APC".JUMP;                                  //save jump input for next call
       #single_previous := "APC".SINGLE;                              //save single input for next call
END_FUNCTION_BLOCK

FUNCTION_BLOCK "AM_BY"   // FB201, SCL
{ S7_Optimized_Access := 'FALSE' }
VERSION : 0.0
// --------------------------------------------------------------------------------
//     program     :    AM_BY
//     description :    apc body module  
//     name        :    D. Bruess
//     date        :    25.11.99
//     
//     revision    :    change default rotation direction: xtal= ccw and cruc= cw
//     name        :    G. Eibelsh鋟ser
//     date        :    26.04.00
// 
//     revision    :    
//     name        :    
//     date        :    
//                     (c)CGS
//     --------------------------------------------------------------------------------
   VAR_INPUT
      start : Bool;   // start sequence, activate step 10 (impulse triggered)
   END_VAR
   VAR
      start_previous : Bool;   // start input value of last call
      cont_previous : Bool;   // cont input value of last call
      resume_previous : Bool;   // resume input value of last call
      jump_previous : Bool;   // jump input value of last call
      single_previous : Bool;   // single input value of last call
      active_step : Array[0..7] of Int;   // active step number for sequence level 0..7
      next_step : Array[0..7] of Int;   // next step number for sequence level 0..7
      hold_step : Array[0..7] of Int;   // step number of step on hold
      end_of_step : Array[0..7] of Bool;   // active step is done flag for sequence 0..7
      EndOfStep : Bool;   // default value for active step is done flag
      cont_enable : Array[0..7] of Bool;   // enable continue function
      ContEnable : Bool;   // default value for enable continue function
      dc_xt_lft_up_prv : Bool;
      dc_cr_lft_up_prv : Bool;
      xt_pos_at_start : Real;   // crystal position at start of body
      set_body_length : Real;   // setpoint body length
   END_VAR
BEGIN


       "APC".STATUS := "APC".BODY;                                     // set apc status               

       "AM_SEQUENCE_CTL" (start_p            := #start,               // control sequence
                        start_previous_p   := #start_previous,
                        cont_previous_p    := #cont_previous, 
                        resume_previous_p  := #resume_previous,
                        jump_previous_p    := #jump_previous,
                        single_previous_p  := #single_previous,
                        active_step_p      := #active_step, 
                        next_step_p        := #next_step,
                        hold_step_p        := #hold_step, 
                        end_of_step_p      := #end_of_step, 
                        cont_enable_p      := #cont_enable); 

       //Set the "Oxidation valve" in all Phases
       "DC".V21_OP:= DINT_TO_BOOL(REAL_TO_DINT("PAR_MAIN".BY_V21_OPEN));

       CASE #active_step[0] OF    //sequence level_0
   //step--0-----level--0-------------------------------------------------off--(sequence off)--------------
           0    :                                                  
                #next_step[0] := 0;

   //step--1-----level--0-------------------------------------------------hold-(test sequence)-------------
           1   :                                                       
               IF #next_step[0] = #active_step[0] THEN                   //init step     
                   //init code
                   ; 
               END_IF;

               //step code                                             //do step
               ;

   //-step-10----level--0----------------------------------------------main-(start sequence)---------------                                                 

   //-step-10----level--0-------------------------------------------------------------                                                 
   //            BY: init body sequence
   //---------------------------------------------------------------------------------                                                 
           10  :                                                     

               // init vacuum system
               // ------------------
               "DC".V1_OP    := TRUE;                         // open V1
               "DC".V3_OP    := FALSE;
               "DC".V4_OP    := FALSE;
               "DC".V5_OP    := TRUE;                         // open V5
               "DC".V6_OP    := FALSE;
               "DC".V8_OP    := FALSE;
               "DC".V11_OP   := FALSE;
               "DC".V11_CL   := TRUE;
               "DC".V12_OP   := FALSE;
               "DC".V13_OP   := FALSE;
               "DC".V20_OP   := FALSE;
               "DC".V22_OP   := FALSE;
               "DC".V24_OP   := FALSE;
               "DC".P1_ON    := TRUE;                         // start main pump
               "DC".P3_ON    := FALSE;
               "DC".V1_OPEN_REQ   := FALSE;                // only EKZ 2700
               "DC".V1_CLOSE_REQ  := FALSE;
               "DC".V3_4_OP  := FALSE;
               "DC".V1_1_REL := FALSE;

               "DC".V3_2_OP := FALSE;                      // vacuum valve feeder

               // init drives
               // -----------
               "DC".XT_LFT_UP := TRUE;                     // crystal lift up
               "DC".XT_LFT_DN := FALSE;
               "DC".XT_LFT_FST := FALSE;
               "DC".XT_ROT_CW := "BM_ROT_DRV_DIR_DB".ROT_DIR;            //1 = cw
               "DC".XT_ROT_CCW := NOT "BM_ROT_DRV_DIR_DB".ROT_DIR;       //0 = ccw


               "DC".CR_LFT_UP := TRUE;                     // crucible lift up
               "DC".CR_LFT_DN := FALSE;
               "DC".CR_LFT_FST := FALSE;
               "DC".CR_ROT_CW := NOT "BM_ROT_DRV_DIR_DB".ROT_DIR;        //0 = cw
               "DC".CR_ROT_CCW := "BM_ROT_DRV_DIR_DB".ROT_DIR;           //1 = ccw


               "AC".SET_XT_SPD := "KYA".SET_XT_SPD;
               "AC".SET_XT_ROT := "KYA".SET_XT_ROT;
               "AC".SET_CR_SPD := "KYA".SET_CR_SPD;
               "AC".SET_CR_ROT := "KYA".SET_CR_ROT;

               // init heater
               // -----------
               "DC".HTR_1_ON := TRUE;                     // heater on
               "DC".HTR_2_ON := TRUE;
               "DC".HTR_3_ON := FALSE;

               // init magnet
               // -----------
               "DC".MAG_ON := ("AC".SET_MAG_1_CUR > 0.0);                       // magnet on

               "AC".SET_MAG_1_CUR := "KYA".SET_MAG_1_CUR;
               "AC".SET_MAG_2_CUR := "KYA".SET_MAG_RATIO_CUR * "AC".SET_MAG_1_CUR;

               // init control loops
               // ------------------
               "DC".CTL_DIA_ON       := FALSE;                   // all control loops off
               "DC".CTL_GRW_RTE_ON   := FALSE;
               "DC".CTL_PULL_RTE_ON  := FALSE;
               "DC".CTL_CRUC_ROT_ON  := FALSE;
               "DC".CTL_MLT_LVL_ON   := TRUE;
               "DC".CTL_MLT_1_TMP_ON := FALSE;
               "DC".CTL_MLT_2_TMP_ON := FALSE;
               "DC".CTL_MLT_DRIFT_ON := FALSE;
               "DC".CTL_GAP_ON       := FALSE;

               "DC".CTL_HTR_1_TMP_ON := TRUE;              // heater temp loop on
               //  DC.CTL_HTR_2_TMP_ON := TRUE;

               "DC".SET_HTR_1_TMP_ABS := FALSE;            // enable inc functions
               "DC".SET_HTR_2_PWR_ABS := FALSE;


               "DC".CTL_PRS_ON := TRUE;                    // pressure control on

               "DC".CTL_SI_FDR_ON := FALSE;
               "DC".CTL_DOP_FDR_ON := FALSE;

               "DV".CR_ROT_CTL_OFFS_RP   := TRUE;                // enable crucible rotation offset ramping to zero
               "DV".CR_ROT_OFFS_RP_START := TRUE;                // set start flag for crucible rotation offset ramping to zero

               "AC".SET_GRW_RTE := 0.0;
               "AC".SET_MLT_1_TMP := 0.0;
               "AC".SET_MLT_2_TMP := 0.0;

               IF ("PAR_MAIN".BY_LSR_LVL_CTL_ON = 1.0) AND "CNF".CONF_LSR_LVL  THEN
                   "AV".SET_MLT_LVL_LSR  := "CTL".ACT_MLT_LVL; //setpoint melt level is written with actual signal of melt level
               ELSE
                   "AV".SET_MLT_LVL_LSR  := 0.0;
               END_IF;    
               "AC".SET_MLT_LVL_LSR  := "AV".SET_MLT_LVL_LSR;

               // init measurement system
               // -----------------------
               "DC".CAM_ISP_ON   :=  TRUE;          //inspection on
               "DC".CAM_INIT     :=  FALSE;
               "DC".CAM_MLT      :=  FALSE;
               "DC".CAM_DIP      :=  FALSE;
               "DC".CAM_DIA      :=  TRUE;
               "DC".CAM_SEL_1    :=  TRUE;
               "DC".CAM_SEL_2    :=  FALSE;

               "DV".THR_CALC_DISABLED  := TRUE;      //threshold calculation in this step is disabled            

               "DC".LSR_ON := ("PAR_MAIN".BY_LSR_LVL_CTL_ON = 1.0);    // laser on/off
               "DC".MCC_ON := FALSE;                       // melt contact control off
               "DC".MCC_TST_ON := FALSE;

               // init Si feeder system
               // ---------------------
               "DC".SI_FDR_ON := FALSE;                    // feeder off
               "DC".DOP_FDR_ON := FALSE;

               "AC".SET_FDR_SI := 0.0;
               "AC".SET_FDR_DOP := 0.0;

               // init lamp on control cabinet
               // ----------------------------
               "DV".LMP_OR := false;

               // save start position, reset length
               // ---------------------------------
               #xt_pos_at_start := "AV".ACT_XT_POS;
               "AV".ACT_XT_LEN_PRC := 0.0; 
               "AV".ACT_XT_LEN := 0.0;

               // reset values for 2nd Body ramp 
               // ------------------------------
               "AM_BY2_RP_CALC_INC_DB".t := 0.0;
               "AM_BY2_RP_CALC_INC_DB".INC := 0.0;
               "AM_BY2_RP_CALC_INC_DB".INC_SUM := 0.0;
               "AV".XT_LEN_BY2_RP := 0.0;

               //init Si charge weight calculation
               //----------------------------------
               "DV".NEW_SI_CRG_WGT_CALC :=  TRUE;

               // calculate all setpoints 
               // -----------------------
               "AM_PAR_FNC_BY" (act_x_value := 0.0);
               //AC.SET_XT_DIA := PAR_MAIN.BY_XT_DIA;    xt setpoint comes from parameter table
               "AC".SET_XT_DIA := "AV".SET_XT_DIA;

               //request exhaust filter flushing when state is switched from service to process next time
               //----------------------------------------------------------------------------------------
               "DV".SI_FIL_FSH_REQ   :=  TRUE;

               // enable automatic mode
               // ---------------------
               "DC".MOD_AUT_ENB := TRUE;

               #end_of_step[0] := true;                            
               #next_step[0] := 100;


   //-step-100---level--0-------------------------------------------------------------                                                 
   //            BY: wait for automatic mode
   //---------------------------------------------------------------------------------                                                 
           100 :                                                     
               IF #next_step[0] = #active_step[0] THEN
                   "APC".OP_MSG := "OP_MSG".WAIT_FOR_AUTO;                                                  
               END_IF;

               // do not count the length while waiting for automatic
               // ---------------------------------------------------
               #xt_pos_at_start := "AV".ACT_XT_POS;
               "AV".ACT_XT_LEN_PRC := 0.0; 
               "AV".ACT_XT_LEN := 0.0;

               // calculate ratio
               // ---------------
               "AV".CRUC_RATIO := "CM_CRUC_RATIO"();

               // calculate all setpoints 
               // -----------------------
               "AM_PAR_FNC_BY" (act_x_value := 0.0);
               //AC.SET_XT_DIA := PAR_MAIN.BY_XT_DIA;   xt setpoint comes from parameter table
               "AC".SET_XT_DIA := "AV".SET_XT_DIA;
               IF "APC".AUTOMATIC = TRUE THEN                     // automatic mode ?
                   #end_of_step[0] := true;                            
               END_IF;                                    
               #next_step[0] := 200;


   //-step-200---level--0-------------------------------------------------------------                                                 
   //            BY: start time
   //---------------------------------------------------------------------------------                                                 
           200 :                                                     
               "APC".ACT_TME_PROC := 0;                           // start process time
               "APC".ACT_TME_STE := 0;                            // reset time of step
               "APC".TI[0] := 0;                                  // start waiting time
               "APC".OP_MSG := "OP_MSG".BLANK;                                                  

               #end_of_step[0] := true;                            
               #next_step[0] := 300;


   //-step-300---level--0-------------------------------------------------------------                                                 
   //            BY: do initial temp. inc.
   //---------------------------------------------------------------------------------                                                 
           300 :                                                     
               IF #next_step[0] = #active_step[0] THEN                       
                   //display initial temperature and power setpoints
                   //-----------------------------------------------
                   "DIS".HTR_1_TMP_SET_PHA_STR   :=  "CTL".SET_HTR_1_TMP;
                   "DIS".HTR_2_PWR_SET_PHA_STR   :=  "CTL".SET_HTR_2_PWR;
                   // do heater inc.
                   // --------------
                   "DC".RSTRT_HTR_1_TMP_INC := TRUE;
                   "DC".RSTRT_HTR_2_PWR_INC := TRUE;
                   "AC".SET_HTR_1_TMP_INC := "AV".SET_HTR_1_TMP_INC;
                   "AC".SET_HTR_2_PWR_INC := "AV".SET_HTR_2_PWR_INC;
               END_IF;

               // calculate actual length
               // -----------------------
               IF ("APC".BYRST) THEN
                   #set_body_length := "AV".SET_XT_LEN_BDY2;        // 2nd body
               ELSE
                   #set_body_length := "PAR_MAIN".BY_XT_LEN;
               END_IF;
               "AM_CALC_LENGTH" (start_pos := #xt_pos_at_start,
                               actual_pos := "AV".ACT_XT_POS,
                               total_len := #set_body_length,
                               actual_len => "AV".ACT_XT_LEN,
                               actual_len_prc => "AV".ACT_XT_LEN_PRC);

               // calculate ratio
               // ---------------
               "AV".CRUC_RATIO := "CM_CRUC_RATIO"();

               // calculate all setpoints for this step
               // ------------------------------------- 
               IF ("APC".BYRST) THEN                          //2nd body                
                   "AM_BY2_RP"();               
                   "AM_PAR_FNC_BY" (act_x_value := "AV".XT_LEN_BY2_RP);
               ELSE          
                   "AM_PAR_FNC_BY" (act_x_value := "AV".ACT_XT_LEN);
               END_IF;                                                 

               "AC".SET_XT_DIA := "AV".SET_XT_DIA;
               "AC".SET_XT_SPD := "AC".SET_AVG_SPD;        // init output diam. control

               // setpoint magnet
               // ---------------
               "DC".MAG_ON := ("AC".SET_MAG_1_CUR > 0.0);

               "AC".SET_MAG_1_CUR := "AV".SET_MAG_1_CUR;
               "AC".SET_MAG_2_CUR := "AC".SET_MAG_RATIO_CUR * "AV".SET_MAG_1_CUR;

               //calculate setpoint melt level
               //-----------------------------
               IF ("PAR_MAIN".BY_LSR_LVL_CTL_ON = 1.0) AND "CNF".CONF_LSR_LVL  THEN
                   "AC".SET_MLT_LVL_LSR  := "AV".SET_MLT_LVL_LSR + "AC".SET_MLT_LVL_INC;
               END_IF;    

               // wait time ?
               // -----------
               IF ("APC".TI[0] > (REAL_TO_INT("PAR_MAIN".BY_DIA_CTRL_ON_DLY))) THEN
                  #end_of_step[0] := true;
               END_IF;

               #next_step[0] := 400; 

   //-step-400---level--0-------------------------------------------------------------                                                 
   //            BY: do body process
   //---------------------------------------------------------------------------------                                                 
           400 :                                                  
               IF #next_step[0] = #active_step[0] THEN                       
                   // diameter and av. speed control on
                   // ---------------------------------
                   "DC".CTL_DIA_ON := TRUE;
                   "DC".CTL_PULL_RTE_ON := TRUE;
               END_IF;
               //set flag for crucible rotation control
               //--------------------------------------
               "DC".CTL_CRUC_ROT_ON := "PAR_MAIN".BY_CRUC_ROT_CTL_ON = 1.0;
               "DV".TRANS_SH_BY_FLAG := FALSE;

               //switch on melt drift control
               //----------------------------
               //DC.CTL_MLT_DRIFT_ON :=  DV.CTL_MLT_DRIFT_ON;

               //read body length from recipe or caluculation
               //--------------------------------------------
               IF ("APC".BYRST) THEN
                   #set_body_length := "AV".SET_XT_LEN_BDY2;        // 2nd body
               ELSE
                   #set_body_length := "PAR_MAIN".BY_XT_LEN;
               END_IF;

               // calculate actual length when offset speed control is on and gap control activated
               // ---------------------------------------------------------------------------------
               IF (("CNF".ACT_DVC_CNF AND 2#0100_0000_0000_0000_0000_0000_0000_0000) = 2#0100_0000_0000_0000_0000_0000_0000_0000) THEN
                   // Calculate crystal length from crystal lift speed set point
                   //-----------------------------------------------------------
                   IF "SysTick100ms" THEN
                       "AV".ACT_XT_LEN:= "AV".ACT_XT_LEN + ("CTL".SET_XT_SPD * 1/600.0);

                       //calc length percentage value
                       //----------------------------
                       IF (#set_body_length > 0.0) THEN
                           "AV".ACT_XT_LEN_PRC:= ("AV".ACT_XT_LEN / #set_body_length) * 100.0;
                       END_IF;
                   END_IF;

                   //set drive direction flags
                   //-------------------------
                   //Set direction of crystal lift
                   //-----------------------------
                   IF (("CTL".SET_XT_SPD + "AV".MLT_LVL_SFT_OFFS_SPD + "CTL".SET_SPEED_OFFS) < 0.0) THEN
                       "DC".XT_LFT_UP    := FALSE;
                       "DC".XT_LFT_DN    := TRUE; // crystal lift down
                       "LT".XT_LFT_UP    := FALSE;
                   ELSE
                       "DC".XT_LFT_UP    := TRUE; // crystal lift up
                       "DC".XT_LFT_DN    := FALSE;
                       "LT".XT_LFT_DN    := FALSE;
                   END_IF;
                   //Set direction of crucible lift
                   //------------------------------
                   IF (("CTL".SET_CR_SPD + "AV".MLT_LVL_SFT_OFFS_SPD + "CTL".SET_SPEED_OFFS ) < 0.0) THEN
                       "DC".CR_LFT_UP    := FALSE;
                       "DC".CR_LFT_DN    := TRUE; // Crucible lift down
                       "LT".CR_LFT_UP    := FALSE;
                   ELSE
                       "DC".CR_LFT_UP    := TRUE; // Crucible lift up
                       "DC".CR_LFT_DN    := FALSE;
                       "LT".CR_LFT_DN    := FALSE;
                   END_IF;

                   //built variables used for manual direction change
                   //------------------------------------------------
                   "DV".MAN_XT_LFT_UP    :=  "DC".XT_LFT_UP AND NOT #dc_xt_lft_up_prv;
                   "DV".MAN_CR_LFT_UP    :=  "DC".CR_LFT_UP AND NOT #dc_cr_lft_up_prv;
                   //store current state of control variables
                   //----------------------------------------
                   #dc_xt_lft_up_prv    :=  "DC".XT_LFT_UP;
                   #dc_cr_lft_up_prv    :=  "DC".CR_LFT_UP;

               // calculate actual length when gap control is deactivated
               // -------------------------------------------------------
               ELSE
                   "AM_CALC_LENGTH" (start_pos := #xt_pos_at_start,
                                   actual_pos := "AV".ACT_XT_POS,
                                   total_len := #set_body_length,
                                   actual_len => "AV".ACT_XT_LEN,
                                   actual_len_prc => "AV".ACT_XT_LEN_PRC);
               END_IF;

               // calculate ratio
               // ---------------
               "AV".CRUC_RATIO := "CM_CRUC_RATIO"();

               // calculate all setpoints for this step
               // -------------------------------------                                      
               IF ("APC".BYRST) THEN                          //2nd body                               
                   "AM_BY2_RP"();
                   "AM_PAR_FNC_BY" (act_x_value := "AV".XT_LEN_BY2_RP);    // set calculated length from 2nd body ramp fnc as body length
               ELSE          
                   "AM_PAR_FNC_BY" (act_x_value := "AV".ACT_XT_LEN);
               END_IF;

               "AC".SET_XT_DIA := "AV".SET_XT_DIA;

               // setpoint magnet
               // ---------------
               "DC".MAG_ON := ("AC".SET_MAG_1_CUR > 0.0);

               "AC".SET_MAG_1_CUR := "AV".SET_MAG_1_CUR;
               "AC".SET_MAG_2_CUR := "AV".SET_MAG_RATIO_CUR * "AV".SET_MAG_1_CUR;

               //calculate setpoint melt level
               //-----------------------------
               IF ("PAR_MAIN".BY_LSR_LVL_CTL_ON = 1.0) AND "CNF".CONF_LSR_LVL  THEN
                   "AC".SET_MLT_LVL_LSR  := "AV".SET_MLT_LVL_LSR + "AC".SET_MLT_LVL_INC;
               END_IF;    

               // heater temp/power inc.
               // ----------------------
               "AC".SET_HTR_1_TMP_INC := "AV".SET_HTR_1_TMP_INC;
               "AC".SET_HTR_2_PWR_INC := "AV".SET_HTR_2_PWR_INC;


               // 100% of length reached ?
               // ------------------------
               IF ("AV".ACT_XT_LEN_PRC >= 100.0) THEN    
                   #end_of_step[0] := true;                            
               END_IF;
               #next_step[0] := 500; 


   //-step-500---level--0-------------------------------------------------------------                                                 
   //            BY: start endcone process
   //---------------------------------------------------------------------------------                                                 
           500 :                                                  
               IF #next_step[0] = #active_step[0] THEN
                   "APC".OP_MSG := "OP_MSG".BLANK;
               END_IF;

               "APC".SUTDN := TRUE;                               // endcone with shut down
               "APC".PNBDY := FALSE;                              // no 2nd body

               "DC".MOD_EC := TRUE;                               // switch to endcone 
               #next_step[0] := 500;                             // E N D 



   //---------------------------------------------------------------------------------                                                 
   //-error------level--0---------------------------------------------------(error in level 0)-------------
       ELSE:                                                        
           //error code                                                //do error code
           ;        
   //------------------------------------------------------------------------------------------------------
       END_CASE;

       CASE #active_step[1] OF    //sequence level_1
   //step--0-----level--1-------------------------------------------------off--(sequence off)--------------
           0    :                                                  
                #next_step[1] := 0;

   //step--1-----level--1-------------------------------------------------hold-(test sequence)-------------
           1   :                                                       
               IF #next_step[1] = #active_step[1] THEN                   //init step     
                   //init code
                   ; 
               END_IF;

               //step code                                             //do step
               ;

   //-step-10----level--1----------------------------------------------main-(start sequence)---------------                                                 
           10  :                                                     
               IF #next_step[1] = #active_step[1] THEN                   //init step     
                   //init code 
                   ;                                                  
               END_IF;

